// TIA Portal V17 export
// export: Created 2024-09-02T12:50:18.8800957Z, ExportSetting WithDefaults, DisplayName Totally Integrated Automation Portal, DisplayVersion V17, DisplayName TIA Portal Openness, DisplayVersion V17, DisplayName TIA Portal Version Control Interface, DisplayVersion V17, DisplayName STEP 7 Professional, DisplayVersion V17, DisplayName STEP 7 Safety, DisplayVersion V17, DisplayName WinCC Professional, DisplayVersion V17
DATA_BLOCK "LTLL_InstMainHMI_OP70"   // DB11
TITLE = LTLL_InstMain
{ DB_Accessible_From_OPC_UA := 'FALSE' }
AUTHOR : Siemens
FAMILY : HMI_Lite
NAME : LTLL_InstMain
VERSION : 8.10
// stored: AutoNumber true, DBAccessibleFromOPCUA false, InstanceOfName LTLL_Main_HMI_OP70, InstanceOfType FB
"LTLL_Main_HMI_OP70"
   // VAR
   //    instLTLL_Basic { S7_SetPoint := 'True'} : "LTLL_Basic";
   //    instLTLL_Manual { S7_SetPoint := 'True'} : "LTLL_Manual";
   //    instLTLL_ManualGraph { S7_SetPoint := 'True'} : "LTLL_ManualGraph";
   //    instLTLL_Sinamics { S7_SetPoint := 'True'} : "LTLL_Sinamics";
   //    instLTLL_Motorstarter { S7_SetPoint := 'True'} : "LTLL_Motorstarter";
   //    instLTLL_RFID { S7_SetPoint := 'True'} : "LTLL_RFID";
   //    instLTLL_Cycletime_1 { S7_SetPoint := 'True'} : "LTLL_Cycletime";
   //    instLTLL_Cycletime { S7_SetPoint := 'True'} : "LTLL_Cycletime";
   //    instLTLL_Counter { S7_SetPoint := 'True'} : "LTLL_Counter";
   //    instLTLL_PLCSystemData { S7_SetPoint := 'True'} : "LTLL_PLCSystemData";
   //    instLTLL_Eks { S7_SetPoint := 'True'} : "LTLL_Eks";
   // END_VAR
BEGIN
END_DATA_BLOCK
